FUNCTION_BLOCK FB_Flash
VAR_INPUT
	tFlashTime : TIME;
END_VAR
VAR_OUTPUT
	
END_VAR
VAR
	fbTon1: TON;
	bDout1: INT;
END_VAR

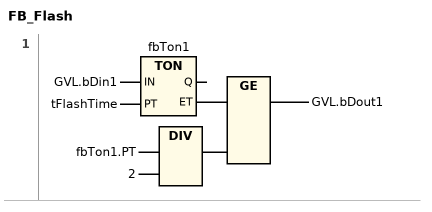
// NETWORK 1
fbTon1(IN := GVL.bDin1, PT := tFlashTime); // TON
GVL.bDout1 := fbTon1.ET >= fbTon1.PT / 2;

END_FUNCTION_BLOCK

(* stored: Version 1.1.0.1, ProductVersion 3.1.4024.12
   POU FB_Flash: Id {0bd846fb-cb0d-4c08-9509-e781dbead45d}, SpecialFunc None *)
